{attribute 'qualified_only'}
VAR_GLOBAL CONSTANT
	EscapeBackslash : BOOL;
END_VAR

(* stored: Version 1.1.0.1, ProductVersion 3.1.4024.15
   GVL EventParameters: Id {cf789bca-2ae3-0a18-3e0d-8421419e656f}, ParameterList True *)
